PROGRAM MAIN
VAR
END_VAR

END_PROGRAM

(* stored: Version 1.1.0.1, ProductVersion 3.1.4024.12
   POU MAIN: Id {f3200a6f-3aae-4825-960f-d37717ef684a}, SpecialFunc None *)
